FUNCTION_BLOCK IN_COLOR (* COLOR input from drop-down list *)
  (* Standard: 61499-1; ApplicationDomain: GUI; Function: COLOR input *)
  (* Version 0.2, 2002-05-03, JHC, Rockwell Automation, Made QI IV=true. *)
  (* Version 0.1, 2001-03-04, JHC, Rockwell Automation, Updated documentation. *)
  (* Version 0.0, 1998-12-29, JHC, Rockwell Automation, SRC version *)
  (* Compiler header: package fb.rt.hmi; import java.awt.*; import java.awt.event.*; *)
  (* Compiler Java IBM VisualAge 3.0 *)
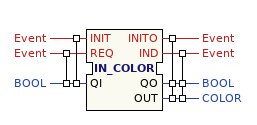
  EVENT_INPUT
    INIT WITH QI; (* Initialization *)
    REQ WITH QI; (* Request *)
  END_EVENT
  EVENT_OUTPUT
    INITO WITH QO, OUT; (* Initialization Confirm *)
    IND WITH QO, OUT; (* User Entered Data or REQ was processed *)
  END_EVENT
  VAR_INPUT
    QI : BOOL := true; (* 1=Read or Init data;0=Inhibit *)
  END_VAR
  VAR_OUTPUT
    QO : BOOL; (* 1=OK,0=Error *)
    OUT : COLOR;
  END_VAR
  SERVICE IN_COLOR/Choice
    SEQUENCE normal_establishment
      IN_COLOR.INIT+() -> Choice.initialize() -> IN_COLOR.INITO+();
    END_SEQUENCE
    SEQUENCE normal_termination
      IN_COLOR.INIT-() -> IN_COLOR.INITO-();
    END_SEQUENCE
    SEQUENCE normal_operation
      Choice.itemStateChanged() -> IN_COLOR.IND+(OUT);
    END_SEQUENCE
    SEQUENCE operation_inhibited
      Choice.itemStateChanged();
    END_SEQUENCE
  END_SERVICE
END_FUNCTION_BLOCK
